FUNCTION_BLOCK ABSTRACT FB_AbstractObservable IMPLEMENTS I_Observable
VAR
    // Dynamic mem
    fbMemMan:                   FB_DynMem_Manager;
    fbBuffer:                   FB_DynMem_Buffer(ipMemMan := fbMemMan);
    pipObserver:                POINTER TO I_Observer;

    aPip:                       ARRAY [0..Param_Observer.cMaxNumberOfObservers-1] OF POINTER TO I_Observer; // Debug array

    // Others
    _bAutoNotify:               BOOL;
END_VAR

METHOD Attach : BOOL
VAR_INPUT
    ipObserver:     I_Observer;
END_VAR
VAR
    i:              UDINT;
END_VAR
// Validate interface pointer
IF ipObserver = 0 THEN
    RETURN;
END_IF

// Max number of observers reached
IF THIS^.nObserverCount >= Param_Observer.cMaxNumberOfObservers THEN
    RETURN;
END_IF

// Create buffer and add observer
IF NOT THIS^.fbBuffer.bAvailable THEN
    THIS^.fbBuffer.CreateBuffer(nSize := SIZEOF(THIS^.pipObserver),
                                bReset := TRUE);

    THIS^.pipObserver := THIS^.fbBuffer.pBuffer;
    THIS^.pipObserver[THIS^.nLastIdx] := ipObserver;
    THIS^.NotifyLast();

    {IF defined(variable: aPip)}
    THIS^.UpdateDebugArray();
    {END_IF}

    Attach := TRUE;
    RETURN;
END_IF

// Make sure observer is not already in the buffer
FOR i := 0 TO THIS^.nLastIdx DO
    IF THIS^.pipObserver[i] = ipObserver THEN
        RETURN;
    END_IF
END_FOR

// Increase buffer size and add observer
THIS^.fbBuffer.Resize(nSize := THIS^.fbBuffer.nBufferSize + SIZEOF(THIS^.pipObserver),
                      bPreserve := TRUE,
                      bReset := FALSE);

THIS^.pipObserver := THIS^.fbBuffer.pBuffer;
THIS^.pipObserver[THIS^.nLastIdx] := ipObserver;
THIS^.NotifyLast();

{IF defined(variable: aPip)}
THIS^.UpdateDebugArray();
{END_IF}

Attach := TRUE;
END_METHOD

METHOD Detach : BOOL
VAR_INPUT
    ipObserver:     I_Observer;
END_VAR
VAR
    i:              UDINT;
    j:              UDINT;
    bFoundItem:     BOOL;
    nRemoveIdx:     UDINT;
    pTmp:           POINTER TO BYTE;
    nPTmpSize:      UDINT;
END_VAR
// Validate interface pointer
IF ipObserver = 0 THEN
    RETURN;
END_IF

// Nothing to remove
IF THIS^.fbBuffer.nBufferSize = 0 THEN
    RETURN;
END_IF

// Find correct observer index to remove
FOR i := 0 TO THIS^.nLastIdx DO
    IF THIS^.pipObserver[i] = ipObserver THEN
        nRemoveIdx := i;
        bFoundItem := TRUE;
        EXIT;
    END_IF
END_FOR

// No item found
IF NOT bFoundItem THEN
    RETURN;

// Found the only item to be removed
ELSIF THIS^.nObserverCount = 1 THEN
    THIS^.fbBuffer.Resize(nSize := 0,
                          bPreserve := FALSE,
                          bReset := TRUE);

    THIS^.pipObserver := THIS^.fbBuffer.pBuffer;

    {IF defined(variable: aPip)}
    THIS^.UpdateDebugArray();
    {END_IF}

    Detach := TRUE;

    RETURN;
END_IF

// Create temporary buffer
nPTmpSize := fbBuffer.nBufferSize - SIZEOF(THIS^.pipObserver);
pTmp := __NEW(BYTE, nPTmpSize);

Tc2_System.MEMCPY(destAddr := pTmp,
                  srcAddr := THIS^.pipObserver,
                  n := nRemoveIdx*SIZEOF(POINTER TO I_Observer));

IF nRemoveIdx < THIS^.nLastIdx THEN
    Tc2_System.MEMCPY(destAddr := pTmp,
                      srcAddr := ADR(THIS^.pipObserver[nRemoveIdx + 1]),
                      n := (THIS^.nLastIdx - nRemoveIdx)*SIZEOF(POINTER TO I_Observer));
END_IF

// Shrink main buffer and clean the contents
THIS^.fbBuffer.Resize(nSize := nPTmpSize,
                      bPreserve := FALSE,
                      bReset := TRUE);

THIS^.pipObserver := fbBuffer.pBuffer;

// Copy contents from temp buffer back to main buffer
Tc2_System.MEMCPY(destAddr := THIS^.pipObserver,
                  srcAddr := pTmp,
                  n := nPTmpSize);

// Delete temp buffer after use
IF pTmp <> 0 THEN
    __DELETE(pTmp);
END_IF

{IF defined(variable: aPip)}
THIS^.UpdateDebugArray();
{END_IF}

Detach := TRUE;
END_METHOD

METHOD FB_init : BOOL
VAR_INPUT
    bInitRetains:       BOOL; // if TRUE, the retain variables are initialized (warm start / cold start)
    bInCopyCode:        BOOL;  // if TRUE, the instance afterwards gets moved into the copy code (online change)
    bAutoNotify:        BOOL;
END_VAR
THIS^._bAutoNotify := bAutoNotify;
END_METHOD

PROPERTY PROTECTED nLastIdx : UDINT
GET
IF THIS^.fbBuffer.nBufferSize > 0 THEN
    nLastIdx := THIS^.fbBuffer.nBufferSize/SIZEOF(THIS^.pipObserver) - 1;
ELSE
    nLastIdx := 0;
END_IF
END_GET
END_PROPERTY

PROPERTY nObserverCount : UDINT
GET
IF THIS^.fbBuffer.nBufferSize > 0 THEN
    nObserverCount := THIS^.nLastIdx + 1;
ELSE
    nObserverCount := 0;
END_IF
END_GET
END_PROPERTY

METHOD ABSTRACT Notify : I_Observable
END_METHOD

METHOD ABSTRACT NotifyLast : I_Observable
END_METHOD

METHOD PRIVATE UpdateDebugArray : BOOL
VAR_INPUT
END_VAR
VAR
    i:                  UDINT;
END_VAR
{IF defined(variable: aPip)}
MEMSET(
    destAddr := ADR(THIS^.aPip),
    fillByte := 0,
    n := SIZEOF(THIS^.aPip));

FOR i := 0 TO THIS^.nLastIdx DO
    THIS^.aPip[i] := ADR(THIS^.pipObserver[i]);
END_FOR
{END_IF}
END_METHOD

END_FUNCTION_BLOCK

(* stored: Version 1.1.0.1, ProductVersion 3.1.4024.12
   POU FB_AbstractObservable: Id {71e23688-66a9-4733-83ac-d64ef266e10a}, SpecialFunc None
   Method Attach: Id {2d2b36e2-7095-4ca4-b111-9d7fc9cde5fd}
   Method Detach: Id {cd87a177-86aa-454f-9754-8649faed008d}
   Method FB_init: Id {cfb9d78b-f9b9-4c25-a6c3-89cdbb34fd0b}
   Property nLastIdx: Id {2c79c953-5622-435d-a939-cc4a5f7e264e}
   Get Get: Id {c29b0475-f6df-4d45-ac76-cc7c5921980f}
   Property nObserverCount: Id {8a1f52c0-3800-483e-a595-61cd3c373210}
   Get Get: Id {11fffc9e-f7b8-44c7-97d9-9f9f0d9e2267}
   Method Notify: Id {50b7b6ea-de79-46bd-bf28-05ba956e9a25}
   Method NotifyLast: Id {bfb98185-9d2f-403d-8101-4e4bed875c91}
   Method UpdateDebugArray: Id {d2dd83c4-e423-4d5c-abb7-4b336ab5b071} *)
